FUNCTION_BLOCK FB_CCA_OOP
VAR_INPUT
	eModeSet :	E_ControlMode := E_ControlMode.Off;	// set control mode
END_VAR
VAR_OUTPUT
	bError					:	BOOL;	
	bInitSuccess			:	BOOL;
END_VAR
VAR
	eModeOld	:	E_ControlMode;

	//Components
	fbHydCir		:	FB_HydMixCirc;
	fbPump			:	FB_PumpBAC_OOP;
	fbValve			:	FB_Valve_2_10V;
	fbTempSupPrim	:	FB_TempSensPt100;
	fbTempRetPrim	:	FB_TempSensPt100;
	fbTempSup		:	FB_TempSensPt100;
	fbTempRet		:	FB_TempSensPt100;
	fbControl		:	FB_CCAController;
END_VAR
VAR_OUTPUT PERSISTENT
		bOperationTestSuccess   : BOOL; 	// True if OperationsTest has been finished sucessfully
		bOperationTestActive 	: BOOL; 	//True if operation test runs
END_VAR

//Initialize if necessary
IF  (eModeOld = E_ControlMode.Off) AND (eModeSet <> E_ControlMode.Off) THEN //Initialize after switching on
	bInitSuccess := FALSE;
END_IF

IF NOT bInitSuccess THEN
	bInitSuccess := Init();
	fbHydCir(iPump := fbPump,
	iValve := fbValve,
	iTempSupPrim := fbTempSupPrim,
	iTempRetPrim := fbTempRetPrim,
	iTempSup := fbTempSup,
	iTempRet := fbTempRet,
	iControl := fbControl,
	eModeSet := eModeSet,
	bInit := TRUE
	);
ELSE
	fbHydCir(iPump := fbPump,
	iValve := fbValve,
	iTempSupPrim := fbTempSupPrim,
	iTempRetPrim := fbTempRetPrim,
	iTempSup := fbTempSup,
	iTempRet := fbTempRet,
	iControl := fbControl,
	eModeSet := eModeSet,
	bInit := FALSE
	);
END_IF

IF fbHydCir.bErr THEN
	bError := TRUE;
ELSE
	bError := FALSE;
END_IF

//write pump info to GVL
PumpInfos.stPumpCCAInfo := fbPump.Info;

//write temperatures to GVL
TempSensors.TempCCASupPrim := fbTempSupPrim.Temperature;
TempSensors.TempCCARetPrim := fbTempRetPrim.Temperature;
TempSensors.TempCCASup := fbTempSup.Temperature;
TempSensors.TempCCARet := fbTempRet.Temperature;

eModeOld := eModeSet;

METHOD Init : BOOL
VAR_INPUT
END_VAR
//Init pump
fbPump.Init();

IF fbPump.InitSuccess AND (NOT fbPump.Error) THEN
	Init := TRUE;
ELSE
	Init := FALSE;
END_IF
END_METHOD

END_FUNCTION_BLOCK

(* stored: Version 1.1.0.1, ProductVersion 3.1.4022.10
   POU FB_CCA_OOP: Id {dad6c183-7fe9-42c9-ab69-8ffe0d7d0677}, SpecialFunc None
   Method Init: Id {573dab19-e8ad-426d-ae2f-93b5734afb73} *)
